// TIA Portal V18 export
VAR_GLOBAL   // PLC tag table "Semafory"
   SV1_red AT %Q14.4 : Bool;
   SV1_yellow AT %Q14.5 : Bool;
   SV1_green AT %Q14.6 : Bool;
   SV2_red AT %Q14.0 : Bool;
   SV2_yellow AT %Q14.1 : Bool;
   SV2_green AT %Q14.2 : Bool;
END_VAR
